INTERFACE I_Disposable EXTENDS T_QueryInterface

// Disposes or release resources for specified task
METHOD Dispose
VAR_INPUT
END_VAR
END_METHOD

END_INTERFACE

(* stored: Version 1.1.0.1, ProductVersion 3.1.4024.4
   Itf I_Disposable: Id {a19faa79-5ada-4236-bfe1-0edd4757a6d2}
   Method Dispose: Id {7997981b-8d5c-4f40-8ae3-54bdda49b7d2} *)
